{attribute 'GeneratedUsingTerminal: KL1644-0050'}
{attribute addProperty BoxType "KL1644-0050"}
{attribute addProperty Description ""}
{attribute addProperty Physics ""}
{attribute addProperty Id "Channel_1AT %Q*Channel_6B723A160Channel_2AT %Q*Channel_6B723A160Channel_3AT %Q*Channel_6B723A160Channel_4AT %Q*Channel_6B723A160"}
{attribute addProperty CRC "1383404149"}
{attribute addProperty Size "0"}
TYPE KL_52751275 :
STRUCT
	{attribute addProperty Name "Channel_1"}
	Channel_1 : Channel_6B723A16;
	{attribute addProperty Name "Channel_2"}
	Channel_2 : Channel_6B723A16;
	{attribute addProperty Name "Channel_3"}
	Channel_3 : Channel_6B723A16;
	{attribute addProperty Name "Channel_4"}
	Channel_4 : Channel_6B723A16;
END_STRUCT
END_TYPE

(* stored: Version 1.2.0.0, ProductVersion 3.1.4024.9
   DUT KL_52751275: Id {90d2e6c4-226a-4982-a096-b558b5e42e3b} *)
